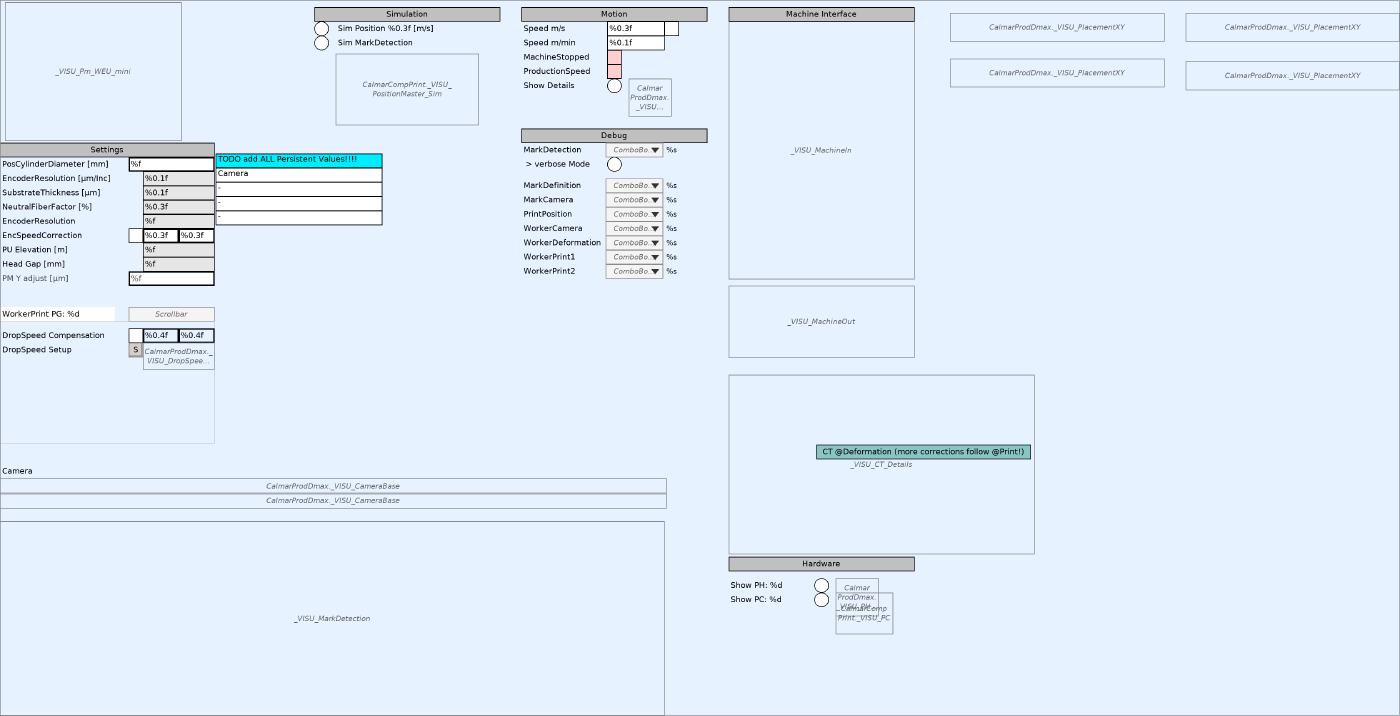
VISUALIZATION _VISU_Pm_WEU_bkp  // 1960x1003
VAR_IN_OUT
  mInst : FB_PrintModule_WEU;
END_VAR
    Rectangle (730,30 120x20), "Speed m/s"
    Rectangle (850,30 80x20), "%0.3f", text variable: mInst.fSpeed
    RoundedRectangle (850,70 20x20), colour toggle: mInst.bMoving
    Rectangle (730,70 110x20), "MachineStopped"
    RoundedRectangle (850,90 20x20), colour toggle: mInst.bProductionSpeedReached
    Rectangle (730,90 110x20), "ProductionSpeed"
    Rectangle (730,50 120x20), "Speed m/min"
    Rectangle (850,50 80x20), "%0.1f", text variable: mInst.fSpeedMpMin
    Rectangle (0,220 180x20), "PosCylinderDiameter [mm]"
    Rectangle (0,240 180x20), "EncoderResolution [µm/Inc]"
    Rectangle (200,240 100x20), "%0.1f", text variable: mInst.fC_EncoderImpU
    Rectangle (180,220 120x20), "%f", text variable: mInst._fEncoderCylinderDiameter
        OnMouseClick: write the text variable via Default
    Rectangle (0,260 180x20), "SubstrateThickness [µm]"
    Rectangle (200,260 100x20), "%0.1f", text variable: mInst._pModuleMachineState^.fSubstrateThickness * 1_000_000
    Rectangle (0,380 180x20), "PM Y adjust [µm]"
    Rectangle (180,380 120x20), "%f", text variable: mInst._fPrintModuleAdjustY
        OnMouseClick: write the text variable via VisuDialogs.Numpad, min PRG_PRINT.sC_Config_P.lL_PU_GENERALSHIFT_Y_SET_MIN, max PRG_PRINT.sC_Config_P.lL_PU_GENERALSHIFT_Y_SET_MAX
    Rectangle (0,360 180x20), "Head Gap [mm]"
    Rectangle (200,360 100x20), "%f", text variable: mInst._pAdsSa^.sI_HeadGap.fI_Val
        OnMouseClick: write the text variable via Default
    RoundedRectangle (930,30 20x20), tooltip "Exeeds max. speed=%f", colour toggle: mInst._pModuleMachineFeedback^.bSpeedExeeded
        p4168582468: mInst._pModuleMachineFeedback^.fMaxSpeed
    Frame (1020,400 260x101)
        shows _VISU_MachineOut(ref := mInst._pModuleMachineFeedback^)
    Frame (1020,30 260x361)
        shows _VISU_MachineIn(ref := mInst._pModuleMachineState^)
    Rectangle (1020,10 260x20), "Machine Interface"
    Rectangle (730,10 260x20), "Motion"
    Frame (0,670 933x22)
        shows CalmarProdDmax._VISU_CameraBase(m_Inst := mInst.fbMarkCameraWeu)
    Frame (0,690 933x22)
        shows CalmarProdDmax._VISU_CameraBase(m_Inst := mInst.fbNoCamera)
    Rectangle (0,650 120x20), "Camera"
    Rectangle (440,10 260x20), "Simulation"
    Ellipse (440,30 20x20), tooltip "Sim position"
        toggle mInst.fbPrintPosition._bSim
    Rectangle (470,30 200x20), "Sim Position %0.3f [m/s]", text variable: mInst.fbPrintPosition.fbPositionMaster._fSimSpeed
        OnMouseClick: write the text variable via Default
    Frame (7,3 247x194)
        shows _VISU_Pm_WEU_mini(mInst := mInst)
    Rectangle (730,110 110x20), "Show Details"
    Ellipse (850,110 20x20)
        toggle mInst.fbView.bShowPositionDetail
    Rectangle (0,200 300x20), "Settings"
    RoundedRectangle (302,235 233x20), "Camera"
    RoundedRectangle (302,255 233x20), "-"
    RoundedRectangle (302,275 233x20), "-"
    RoundedRectangle (302,295 233x20), "-"
    RoundedRectangle (302,215 233x20), "TODO add ALL Persistent Values!!!!"
    Rectangle (250,320 50x20), "%0.3f", tooltip "Encoder speed compensation reference speed", text variable: mInst.fbPrintPosition._fSpeedCompRefSpeed
        OnMouseClick: write the text variable via Default
    Rectangle (200,320 50x20), "%0.3f", tooltip "Encoder speed compensation factor", text variable: mInst.fbPrintPosition._fSpeedCompFactor
        OnMouseClick: write the text variable via Default
    RoundedRectangle (180,320 20x20)
        toggle mInst.fbPrintPosition._bEnSpeedComp
    Rectangle (0,320 180x20), "EncSpeedCorrection"
    Rectangle (0,300 180x20), "EncoderResolution"
    Rectangle (200,300 100x20), "%f", text variable: mInst.fbPrintPosition._fEncoderResolution
    Rectangle (0,280 180x20), "NeutralFiberFactor [%]"
    Rectangle (200,280 100x20), "%0.3f", text variable: mInst._pModuleMachineState^.fNeutralFibreFactor
    Scrollbar (180,430 120x20)
        p2245068023: GVL_WEU.nC_WorkerPrintPerPm
        p1057716461: mInst.fbView.nSelWorkerPrint
    Rectangle (0,430 160x20), "WorkerPrint PG: %d", text variable: mInst.fbView.nSelWorkerPrint
    Rectangle (0,450 300x171)
    Rectangle (0,460 180x20), "DropSpeed Compensation"
    Rectangle (200,460 50x20), "%0.4f", tooltip "DropSpeed [m/s]", text variable: mInst.fbWorkerPrint[mInst.fbView.nSelWorkerPrint].fbDropSpeedComp.fDropSpeed
        OnMouseClick: write the text variable via Default
    Rectangle (250,460 50x20), "%0.4f", tooltip "Dead/Add Time [ms]", text variable: mInst.fbWorkerPrint[mInst.fbView.nSelWorkerPrint].fbDropSpeedComp.fDropSpeedDeadTime
        OnMouseClick: write the text variable via Default
    RoundedRectangle (180,460 20x20), tooltip "Enabled compensation", input disabled if: TRUE
        toggle mInst.fbWorkerPrint[mInst.fbView.nSelWorkerPrint].fbDropSpeedComp._bEnable p2164770859=TRUE
    Button (180,480 20x20), "S", tooltip "Setup"
        toggle minst.fbView.bShowDropSpeedSetup
    Rectangle (0,480 180x20), "DropSpeed Setup"
    Frame (0,730 930x273)
        shows _VISU_MarkDetection(mInst := mInst.fbMarkDetection)
    Ellipse (440,50 20x20), tooltip "Sim position"
        toggle mInst.fbMarkDetection.bSimEnable
    Rectangle (470,50 200x20), "Sim MarkDetection"
    Rectangle (730,180 260x20), "Debug"
    Rectangle (730,200 120x20), "MarkDetection"
    Rectangle (730,250 120x20), "MarkDefinition"
    Rectangle (930,250 60x20), "%s", tooltip "LogLevel", text variable: mInst.fbMarkDefinition._loglevel
        OnMouseClick: write the text variable via Default
    Rectangle (730,270 120x20), "MarkCamera"
    Rectangle (930,270 60x20), "%s", tooltip "LogLevel", text variable: mInst.fbMarkCameraWeu._loglevel
        OnMouseClick: write the text variable via Default
    Rectangle (730,290 120x20), "PrintPosition"
    Rectangle (930,290 60x20), "%s", tooltip "LogLevel", text variable: mInst.fbPrintPosition._loglevel
        OnMouseClick: write the text variable via Default
    Rectangle (730,310 120x20), "WorkerCamera"
    Rectangle (930,310 60x20), "%s", tooltip "LogLevel", text variable: mInst.fbWorkerCamera._loglevel
        OnMouseClick: write the text variable via Default
    Rectangle (730,350 120x20), "WorkerPrint1"
    Rectangle (930,350 60x20), "%s", tooltip "LogLevel", text variable: mInst.fbWorkerPrint[1]._loglevel
        OnMouseClick: write the text variable via Default
    Rectangle (730,370 120x20), "WorkerPrint2"
    Rectangle (930,370 60x20), "%s", tooltip "LogLevel", text variable: mInst.fbWorkerPrint[2]._loglevel
        OnMouseClick: write the text variable via Default
    Frame (200,480 100x38), invisible if: NOT minst.fbView.bShowDropSpeedSetup
        shows CalmarProdDmax._VISU_DropSpeedComp_Setup(mInst := mInst.fbWorkerPrint[mInst.fbView.nSelWorkerPrint].fbDropSpeedComp)
    Frame (880,110 60x53), invisible if: NOT mInst.fbView.bShowPositionDetail
        shows CalmarProdDmax._VISU_PrintPositionDmax(m_Inst := mInst.fbPrintPosition)
    Rectangle (726,220 124x20), "> verbose Mode"
    Ellipse (850,220 20x20)
        toggle mInst.fbMarkDetection._bVerbose
    Frame (1020,525 428x251)
        shows _VISU_CT_Details(mInst := mInst.fbWorkerDeformation)
    Rectangle (730,330 120x20), "WorkerDeformation"
    Rectangle (930,330 60x20), "%s", tooltip "LogLevel", text variable: mInst.fbWorkerDeformation._loglevel
        OnMouseClick: write the text variable via Default
    ComboBoxInteger (848,350 80x20), tooltip "LogLevel", variable: mInst.fbWorkerPrint[1]._loglevel, text list: 'LogSeverity'
    ComboBoxInteger (848,370 80x20), tooltip "LogLevel", variable: mInst.fbWorkerPrint[2]._loglevel, text list: 'LogSeverity'
    ComboBoxInteger (848,330 80x20), tooltip "LogLevel", variable: mInst.fbWorkerDeformation._loglevel, text list: 'LogSeverity'
    ComboBoxInteger (848,310 80x20), tooltip "LogLevel", variable: mInst.fbWorkerCamera._loglevel, text list: 'LogSeverity'
    ComboBoxInteger (848,290 80x20), tooltip "LogLevel", variable: mInst.fbPrintPosition._loglevel, text list: 'LogSeverity'
    ComboBoxInteger (848,270 80x20), tooltip "LogLevel", variable: mInst.fbMarkCameraWeu._loglevel, text list: 'LogSeverity'
    ComboBoxInteger (848,250 80x20), tooltip "LogLevel", variable: mInst.fbMarkDefinition._loglevel, text list: 'LogSeverity'
    Rectangle (930,200 60x20), "%s", tooltip "LogLevel", text variable: mInst.fbMarkDetection._loglevel
        OnMouseClick: write the text variable via Default
    ComboBoxInteger (848,200 80x20), tooltip "LogLevel", variable: mInst.fbMarkDetection._loglevel, text list: 'LogSeverity'
    Ellipse (1140,810 20x20)
        toggle mInst.fbView.bShowPhDetail
    Frame (1170,810 60x53), invisible if: NOT mInst.fbView.bShowPhDetail
        shows CalmarProdDmax._VISU_PH_Grid(m_Inst := mInst._pPh[mInst.fbView.nSelPhDetail]^)
    Rectangle (1020,810 110x20), "Show PH: %d", text variable: mInst.fbView.nSelPhDetail
        OnMouseClick: write the text variable via Default
    Rectangle (1020,780 260x20), "Hardware"
    Ellipse (1140,830 20x20)
        toggle mInst.fbView.bShowPcDetail
    Frame (1170,830 80x58), invisible if: NOT mInst.fbView.bShowPcDetail
        shows CalmarCompPrint._VISU_PC(m_Inst := mInst._pPc[mInst.fbView.nSelPcDetail]^)
    Rectangle (1020,830 110x20), "Show PC: %d", text variable: mInst.fbView.nSelPcDetail
        OnMouseClick: write the text variable via Default
    Rectangle (200,340 100x20), "%f", text variable: mInst.fPuElevation
        OnMouseClick: write the text variable via Default
    Rectangle (0,340 180x20), "PU Elevation [m]"
    Frame (470,75 200x100)
        shows CalmarCompPrint._VISU_PositionMaster_Sim(mInst := mInst.fbPrintPosition.fbPositionMaster)
    Frame (1330,18 300x40)
        shows CalmarProdDmax._VISU_PlacementXY(m_Inst := mInst.fbFineAlignement._fbPUCorrPoints[1])
    Frame (1660,18 300x40)
        shows CalmarProdDmax._VISU_PlacementXY(m_Inst := mInst.fbFineAlignement._fbPUCorrPoints[2])
    Frame (1330,82 300x40)
        shows CalmarProdDmax._VISU_PlacementXY(m_Inst := mInst.fbFineAlignement._fbPUCorrPoints[3])
    Frame (1660,86 300x40)
        shows CalmarProdDmax._VISU_PlacementXY(m_Inst := mInst.fbFineAlignement._fbPUCorrPoints[4])
    Rectangle (1143,623 300x20), "CT @Deformation (more corrections follow @Print!)"
END_VISUALIZATION

(* stored: Version 1.1.0.1, ProductVersion 3.1.4024.11
   Visu _VISU_Pm_WEU_bkp: Id {d684c312-9b46-4054-ba36-c1da46360bb5} *)
